% RSLogix 500 project P1_DLOGIX_BAK002.RSS, saved by version 12.00.00.00 %
PROJECT "UNTITLED"    % processor: Bul.1763 MicroLogix 1100 Series B %

PROGRAM FILES
  LAD 2 "MAIN"  3 rungs
  LAD 4 "DIGITAL IO"  5 rungs
  LAD 5 "CONTROL"  7 rungs

DATA FILES
  O0 OUTPUT  4 elements
  I1 INPUT  6 elements
  S2 STATUS  66 elements
  B3 BINARY  1 elements
  T4 TIMER  4 elements
  C5 COUNTER  1 elements
  R6 CONTROL  1 elements
  N7 INTEGER  1 elements
  F8 FLOAT  1 elements

LADDER 2 "MAIN"
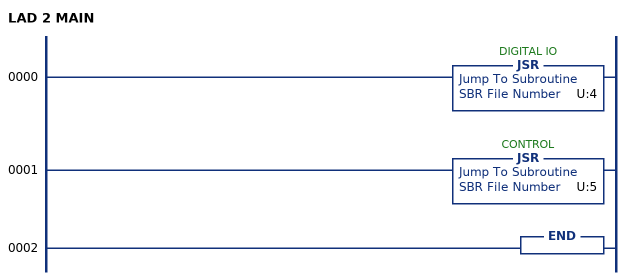
% Rung: 0 %
SOR JSR U:4 EOR
%   U:4  "DIGITAL IO" %
% Rung: 1 %
SOR JSR U:5 EOR
%   U:5  "CONTROL" %
% Rung: 2 %
SOR END EOR

LADDER 4 "DIGITAL IO"
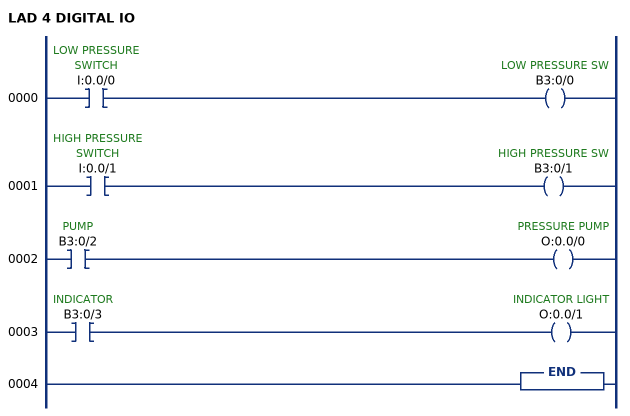
% Rung: 0 %
SOR XIC I:0.0/0 OTE B3:0/0 EOR
%   I:0.0/0  "LOW PRESSURE SWITCH" %
%   B3:0/0  "LOW PRESSURE SW" %
% Rung: 1 %
SOR XIC I:0.0/1 OTE B3:0/1 EOR
%   I:0.0/1  "HIGH PRESSURE SWITCH" %
%   B3:0/1  "HIGH PRESSURE SW" %
% Rung: 2 %
SOR XIC B3:0/2 OTE O:0.0/0 EOR
%   B3:0/2  "PUMP" %
%   O:0.0/0  "PRESSURE PUMP" %
% Rung: 3 %
SOR XIC B3:0/3 OTE O:0.0/1 EOR
%   B3:0/3  "INDICATOR" %
%   O:0.0/1  "INDICATOR LIGHT" %
% Rung: 4 %
SOR END EOR

LADDER 5 "CONTROL"
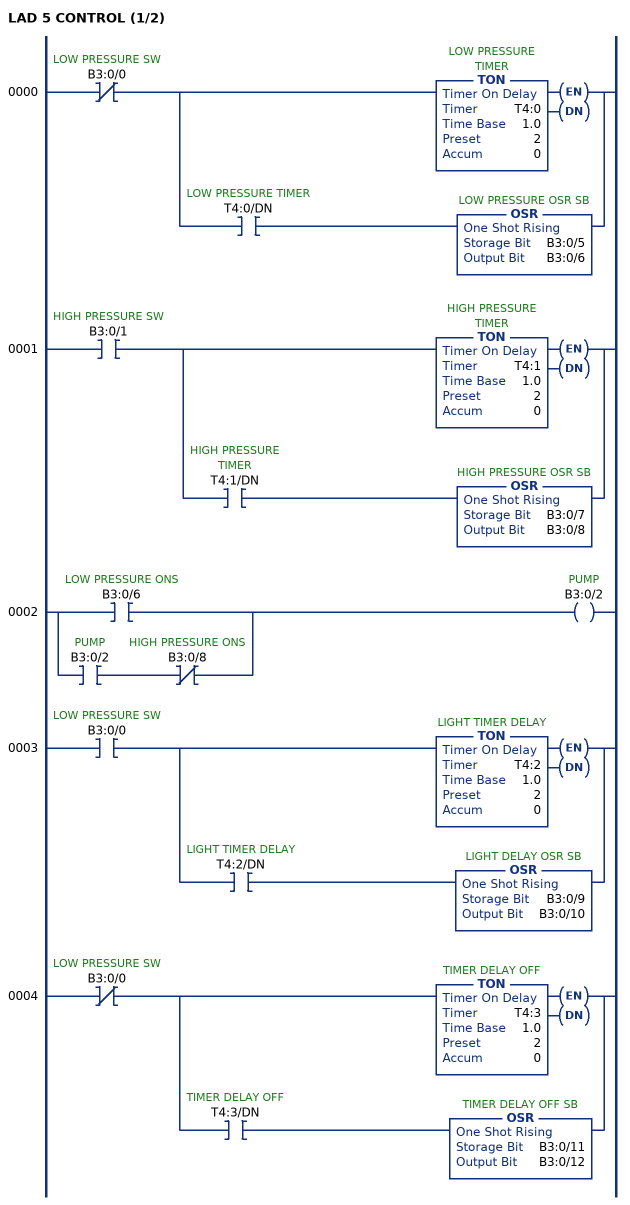
% Rung: 0 %
SOR XIO B3:0/0 BST TON T4:0 1.0 2 0 NXB XIC T4:0/DN OSR B3:0/5 B3:0/6 BND EOR
%   B3:0/0  "LOW PRESSURE SW" %
%   T4:0  "LOW PRESSURE TIMER" %
%   B3:0/5  "LOW PRESSURE OSR SB" %
%   B3:0/6  "LOW PRESSURE ONS" %
% Rung: 1 %
SOR XIC B3:0/1 BST TON T4:1 1.0 2 0 NXB XIC T4:1/DN OSR B3:0/7 B3:0/8 BND EOR
%   B3:0/1  "HIGH PRESSURE SW" %
%   T4:1  "HIGH PRESSURE TIMER" %
%   B3:0/7  "HIGH PRESSURE OSR SB" %
%   B3:0/8  "HIGH PRESSURE ONS" %
% Rung: 2 %  % edit flag set %
SOR BST XIC B3:0/6 NXB XIC B3:0/2 XIO B3:0/8 BND OTE B3:0/2 EOR
%   B3:0/6  "LOW PRESSURE ONS" %
%   B3:0/2  "PUMP" %
%   B3:0/8  "HIGH PRESSURE ONS" %
% Rung: 3 %
SOR XIC B3:0/0 BST TON T4:2 1.0 2 0 NXB XIC T4:2/DN OSR B3:0/9 B3:0/10 BND EOR
%   B3:0/0  "LOW PRESSURE SW" %
%   T4:2  "LIGHT TIMER DELAY" %
%   B3:0/9  "LIGHT DELAY OSR SB" %
%   B3:0/10  "TIMER DELAY OSR" %
% Rung: 4 %
SOR XIO B3:0/0 BST TON T4:3 1.0 2 0 NXB XIC T4:3/DN OSR B3:0/11 B3:0/12 BND EOR
%   B3:0/0  "LOW PRESSURE SW" %
%   T4:3  "TIMER DELAY OFF" %
%   B3:0/11  "TIMER DELAY OFF SB" %
%   B3:0/12  "TIMER DEALY OFF OSR" %

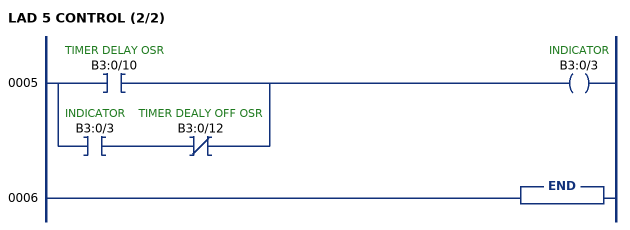
% Rung: 5 %
SOR BST XIC B3:0/10 NXB XIC B3:0/3 XIO B3:0/12 BND OTE B3:0/3 EOR
%   B3:0/10  "TIMER DELAY OSR" %
%   B3:0/3  "INDICATOR" %
%   B3:0/12  "TIMER DEALY OFF OSR" %
% Rung: 6 %
SOR END EOR

OTHER DOCUMENTED ADDRESSES
  B3:0/4  "PUMP CONTROL 0= PUMP OFF 1= PUMP ON"

DATA TABLE (non-zero values as saved)
DATA T4
% .PRE .ACC %
% T4:0 % 2 0
% T4:1 % 2 0
% T4:2 % 2 0
% T4:3 % 2 0
